Fanuc TP program (LS listing): DISTI_CADC_V5.LS

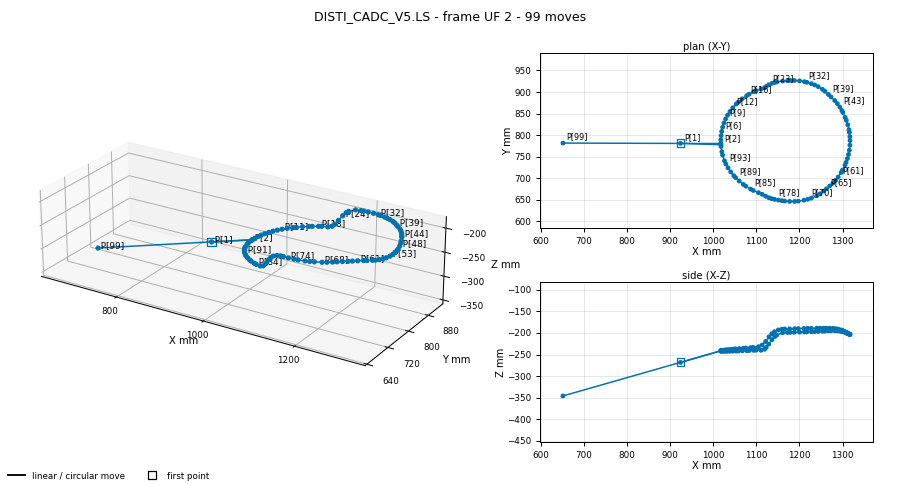
[picture p0: tool path of DISTI_CADC_V5.LS in frame UF 2, 99 of 99 moves have a stored position in this frame; points joined in program order, loops and branches not executed]
/PROG  DISTI_CADC_V5
/ATTR
OWNER		= MNEDITOR;
COMMENT		= "WeldPRO Auto-Gen";
PROG_SIZE	= 7125;
CREATE		= DATE 26-07-30  TIME 16:50:06;
MODIFIED	= DATE 26-07-30  TIME 17:29:32;
FILE_NAME	= DISTI_CA;
VERSION		= 0;
LINE_COUNT	= 113;
MEMORY_SIZE	= 7445;
PROTECT		= READ_WRITE;
TCD:  STACK_SIZE	= 0,
      TASK_PRIORITY	= 50,
      TIME_SLICE	= 0,
      BUSY_LAMP_OFF	= 0,
      ABORT_REQUEST	= 0,
      PAUSE_REQUEST	= 0;
DEFAULT_GROUP	= 1,*,*,*,*;
CONTROL_CODE	= 00000000 00000000;
/APPL
/MN
   1:  !WeldPRO Auto-Generated TPP ;
   2:  !TOR_XL_2026, TOR_xl_2907 ;
   3:   ;
   4:  UFRAME_NUM=2 ;
   5:  UTOOL_NUM=2 ;
   6:  !Feature Approach ;
   7:J P[1] 100% FINE    ;
   8:   ;
   9:  !Segment1 ;
  10:L P[2] 2000mm/sec FINE    ;
  11:   ;
  12:  CALL LASER_OFF    ;
  13:L P[3] R[23:moving]mm/sec CNT100    ;
  14:L P[4] R[23:moving]mm/sec CNT100    ;
  15:L P[5] R[23:moving]mm/sec CNT100    ;
  16:L P[6] R[23:moving]mm/sec CNT100    ;
  17:L P[7] R[23:moving]mm/sec CNT100    ;
  18:L P[8] R[23:moving]mm/sec CNT100    ;
  19:L P[9] R[23:moving]mm/sec CNT100    ;
  20:L P[10] R[23:moving]mm/sec CNT100    ;
  21:L P[11] R[23:moving]mm/sec CNT100    ;
  22:L P[12] R[23:moving]mm/sec CNT100    ;
  23:L P[13] R[23:moving]mm/sec CNT100    ;
  24:L P[14] R[23:moving]mm/sec CNT100    ;
  25:L P[15] R[23:moving]mm/sec CNT100    ;
  26:L P[16] R[23:moving]mm/sec CNT100    ;
  27:L P[17] R[23:moving]mm/sec CNT100    ;
  28:L P[18] R[23:moving]mm/sec CNT100    ;
  29:L P[19] R[23:moving]mm/sec CNT100    ;
  30:L P[20] R[23:moving]mm/sec CNT100    ;
  31:L P[21] R[23:moving]mm/sec CNT100    ;
  32:L P[22] R[23:moving]mm/sec CNT100    ;
  33:L P[23] R[23:moving]mm/sec CNT100    ;
  34:L P[24] R[23:moving]mm/sec CNT100    ;
  35:L P[25] R[23:moving]mm/sec CNT100    ;
  36:L P[26] R[23:moving]mm/sec CNT100    ;
  37:L P[27] R[23:moving]mm/sec CNT100    ;
  38:L P[28] R[23:moving]mm/sec CNT100    ;
  39:L P[29] R[23:moving]mm/sec CNT100    ;
  40:L P[30] R[23:moving]mm/sec CNT100    ;
  41:L P[31] R[23:moving]mm/sec CNT100    ;
  42:L P[32] R[23:moving]mm/sec CNT100    ;
  43:L P[33] R[23:moving]mm/sec CNT100    ;
  44:L P[34] R[23:moving]mm/sec CNT100    ;
  45:L P[35] R[23:moving]mm/sec CNT100    ;
  46:L P[36] R[23:moving]mm/sec CNT100    ;
  47:L P[37] R[23:moving]mm/sec CNT100    ;
  48:L P[38] R[23:moving]mm/sec CNT100    ;
  49:L P[39] R[23:moving]mm/sec CNT100    ;
  50:L P[40] R[23:moving]mm/sec CNT100    ;
  51:L P[41] R[23:moving]mm/sec CNT100    ;
  52:L P[42] R[23:moving]mm/sec CNT100    ;
  53:L P[43] R[23:moving]mm/sec CNT100    ;
  54:L P[44] R[23:moving]mm/sec CNT100    ;
  55:L P[45] R[23:moving]mm/sec CNT100    ;
  56:L P[46] R[23:moving]mm/sec CNT100    ;
  57:L P[47] R[23:moving]mm/sec CNT100    ;
  58:L P[48] R[23:moving]mm/sec CNT100    ;
  59:L P[49] R[23:moving]mm/sec CNT100    ;
  60:L P[50] R[23:moving]mm/sec CNT100    ;
  61:L P[51] R[23:moving]mm/sec CNT100    ;
  62:L P[52] R[23:moving]mm/sec CNT100    ;
  63:L P[53] R[23:moving]mm/sec CNT100    ;
  64:L P[54] R[23:moving]mm/sec CNT100    ;
  65:L P[55] R[23:moving]mm/sec CNT100    ;
  66:L P[56] R[23:moving]mm/sec CNT100    ;
  67:L P[57] R[23:moving]mm/sec CNT100    ;
  68:L P[58] R[23:moving]mm/sec CNT100    ;
  69:L P[59] R[23:moving]mm/sec CNT100    ;
  70:L P[60] R[23:moving]mm/sec CNT100    ;
  71:L P[61] R[23:moving]mm/sec CNT100    ;
  72:L P[62] R[23:moving]mm/sec CNT100    ;
  73:L P[63] R[23:moving]mm/sec CNT100    ;
  74:L P[64] R[23:moving]mm/sec CNT100    ;
  75:L P[65] R[23:moving]mm/sec CNT100    ;
  76:L P[66] R[23:moving]mm/sec CNT100    ;
  77:L P[67] R[23:moving]mm/sec CNT100    ;
  78:L P[68] R[23:moving]mm/sec CNT100    ;
  79:L P[69] R[23:moving]mm/sec CNT100    ;
  80:L P[70] R[23:moving]mm/sec CNT100    ;
  81:L P[71] R[23:moving]mm/sec CNT100    ;
  82:L P[72] R[23:moving]mm/sec CNT100    ;
  83:L P[73] R[23:moving]mm/sec CNT100    ;
  84:L P[74] R[23:moving]mm/sec CNT100    ;
  85:L P[75] R[23:moving]mm/sec CNT100    ;
  86:L P[76] R[23:moving]mm/sec CNT100    ;
  87:L P[77] R[23:moving]mm/sec CNT100    ;
  88:L P[78] R[23:moving]mm/sec CNT100    ;
  89:L P[79] R[23:moving]mm/sec CNT100    ;
  90:L P[80] R[23:moving]mm/sec CNT100    ;
  91:L P[81] R[23:moving]mm/sec CNT100    ;
  92:L P[82] R[23:moving]mm/sec CNT100    ;
  93:L P[83] R[23:moving]mm/sec CNT100    ;
  94:L P[84] R[23:moving]mm/sec CNT100    ;
  95:L P[85] R[23:moving]mm/sec CNT100    ;
  96:L P[86] R[23:moving]mm/sec CNT100    ;
  97:L P[87] R[23:moving]mm/sec CNT100    ;
  98:L P[88] R[23:moving]mm/sec CNT100    ;
  99:L P[89] R[23:moving]mm/sec CNT100    ;
 100:L P[90] R[23:moving]mm/sec CNT100    ;
 101:L P[91] R[23:moving]mm/sec CNT100    ;
 102:L P[92] R[23:moving]mm/sec CNT100    ;
 103:L P[93] R[23:moving]mm/sec CNT100    ;
 104:L P[94] R[23:moving]mm/sec CNT100    ;
 105:L P[95] R[23:moving]mm/sec CNT100    ;
 106:L P[96] R[23:moving]mm/sec CNT100    ;
 107:L P[97] R[23:moving]mm/sec CNT100    ;
 108:L P[98] R[23:moving]mm/sec FINE    ;
 109:  CALL LASER_OFF    ;
 110:   ;
 111:  !Feature Retreat ;
 112:L P[99] 2000mm/sec FINE    ;
 113:  CALL ROTATE    ;
/POS
P[1]{
   GP1:
	UF : 2, UT : 2,		CONFIG : 'F D T, 0, 0, 0',
	X =   924.335  mm,	Y =   780.986  mm,	Z =  -268.284  mm,
	W =  -106.495 deg,	P =   -15.000 deg,	R =    94.234 deg
};
P[2]{
   GP1:
	UF : 2, UT : 2,		CONFIG : 'F D T, 0, 0, 0',
	X =  1018.100  mm,	Y =   777.871  mm,	Z =  -241.295  mm,
	W =  -106.497 deg,	P =   -14.995 deg,	R =    94.216 deg
};
P[3]{
   GP1:
	UF : 2, UT : 2,		CONFIG : 'F D T, 0, 0, 0',
	X =  1017.949  mm,	Y =   780.606  mm,	Z =  -241.391  mm,
	W =  -106.499 deg,	P =   -14.997 deg,	R =    94.226 deg
};
P[4]{
   GP1:
	UF : 2, UT : 2,		CONFIG : 'F D T, 0, 0, 0',
	X =  1017.881  mm,	Y =   789.004  mm,	Z =  -241.645  mm,
	W =  -106.492 deg,	P =   -15.098 deg,	R =    90.372 deg
};
P[5]{
   GP1:
	UF : 2, UT : 2,		CONFIG : 'F D T, 0, 0, 0',
	X =  1018.505  mm,	Y =   798.964  mm,	Z =  -241.908  mm,
	W =  -106.481 deg,	P =   -15.218 deg,	R =    85.605 deg
};
P[6]{
   GP1:
	UF : 2, UT : 2,		CONFIG : 'F D T, 0, 0, 0',
	X =  1019.837  mm,	Y =   808.597  mm,	Z =  -242.115  mm,
	W =  -106.456 deg,	P =   -15.335 deg,	R =    80.815 deg
};
P[7]{
   GP1:
	UF : 2, UT : 2,		CONFIG : 'F D T, 0, 0, 0',
	X =  1022.039  mm,	Y =   818.579  mm,	Z =  -242.280  mm,
	W =  -106.423 deg,	P =   -15.450 deg,	R =    76.090 deg
};
P[8]{
   GP1:
	UF : 2, UT : 2,		CONFIG : 'F D T, 0, 0, 0',
	X =  1025.052  mm,	Y =   828.219  mm,	Z =  -242.385  mm,
	W =  -106.378 deg,	P =   -15.565 deg,	R =    71.217 deg
};
P[9]{
   GP1:
	UF : 2, UT : 2,		CONFIG : 'F D T, 0, 0, 0',
	X =  1028.881  mm,	Y =   837.505  mm,	Z =  -242.427  mm,
	W =  -106.322 deg,	P =   -15.679 deg,	R =    66.207 deg
};
P[10]{
   GP1:
	UF : 2, UT : 2,		CONFIG : 'F D T, 0, 0, 0',
	X =  1033.533  mm,	Y =   846.438  mm,	Z =  -242.409  mm,
	W =  -106.254 deg,	P =   -15.791 deg,	R =    61.015 deg
};
P[11]{
   GP1:
	UF : 2, UT : 2,		CONFIG : 'F D T, 0, 0, 0',
	X =  1038.975  mm,	Y =   854.961  mm,	Z =  -242.328  mm,
	W =  -106.177 deg,	P =   -15.894 deg,	R =    55.979 deg
};
P[12]{
   GP1:
	UF : 2, UT : 2,		CONFIG : 'F D T, 0, 0, 0',
	X =  1045.527  mm,	Y =   863.473  mm,	Z =  -242.178  mm,
	W =  -106.096 deg,	P =   -15.986 deg,	R =    51.162 deg
};
P[13]{
   GP1:
	UF : 2, UT : 2,		CONFIG : 'F D T, 0, 0, 0',
	X =  1053.550  mm,	Y =   872.150  mm,	Z =  -241.942  mm,
	W =  -106.012 deg,	P =   -16.066 deg,	R =    46.632 deg
};
P[14]{
   GP1:
	UF : 2, UT : 2,		CONFIG : 'F D T, 0, 0, 0',
	X =  1058.278  mm,	Y =   876.579  mm,	Z =  -241.784  mm,
	W =  -105.919 deg,	P =   -16.142 deg,	R =    41.952 deg
};
P[15]{
   GP1:
	UF : 2, UT : 2,		CONFIG : 'F D T, 0, 0, 0',
	X =  1067.621  mm,	Y =   884.365  mm,	Z =  -241.434  mm,
	W =  -105.870 deg,	P =   -16.177 deg,	R =    39.609 deg
};
P[16]{
   GP1:
	UF : 2, UT : 2,		CONFIG : 'F D T, 0, 0, 0',
	X =  1077.833  mm,	Y =   891.592  mm,	Z =  -241.014  mm,
	W =  -105.777 deg,	P =   -16.235 deg,	R =    35.365 deg
};
P[17]{
   GP1:
	UF : 2, UT : 2,		CONFIG : 'F D T, 0, 0, 0',
	X =  1083.331  mm,	Y =   894.952  mm,	Z =  -240.778  mm,
	W =  -105.677 deg,	P =   -16.289 deg,	R =    30.964 deg
};
P[18]{
   GP1:
	UF : 2, UT : 2,		CONFIG : 'F D T, 0, 0, 0',
	X =  1094.066  mm,	Y =   900.628  mm,	Z =  -240.278  mm,
	W =  -105.579 deg,	P =   -16.333 deg,	R =    26.830 deg
};
P[19]{
   GP1:
	UF : 2, UT : 2,		CONFIG : 'F D T, 0, 0, 0',
	X =  1099.603  mm,	Y =   903.126  mm,	Z =  -240.005  mm,
	W =  -105.536 deg,	P =   -16.344 deg,	R =    25.018 deg
};
P[20]{
   GP1:
	UF : 2, UT : 2,		CONFIG : 'F D T, 0, 0, 0',
	X =  1111.079  mm,	Y =   907.027  mm,	Z =  -240.106  mm,
	W =  -116.027 deg,	P =   -16.063 deg,	R =    30.267 deg
};
P[21]{
   GP1:
	UF : 2, UT : 2,		CONFIG : 'F D T, 0, 0, 0',
	X =  1119.171  mm,	Y =   909.914  mm,	Z =  -237.723  mm,
	W =  -126.877 deg,	P =   -15.356 deg,	R =    25.893 deg
};
P[22]{
   GP1:
	UF : 2, UT : 2,		CONFIG : 'F D T, 0, 0, 0',
	X =  1122.964  mm,	Y =   912.740  mm,	Z =  -233.580  mm,
	W =  -119.393 deg,	P =   -15.981 deg,	R =    16.221 deg
};
P[23]{
   GP1:
	UF : 2, UT : 2,		CONFIG : 'F D T, 0, 0, 0',
	X =  1128.743  mm,	Y =   916.697  mm,	Z =  -225.925  mm,
	W =  -115.329 deg,	P =   -16.208 deg,	R =    11.788 deg
};
P[24]{
   GP1:
	UF : 2, UT : 2,		CONFIG : 'F D T, 0, 0, 0',
	X =  1136.345  mm,	Y =   920.133  mm,	Z =  -215.586  mm,
	W =  -112.639 deg,	P =   -16.315 deg,	R =     9.714 deg
};
P[25]{
   GP1:
	UF : 2, UT : 2,		CONFIG : 'F D T, 0, 0, 0',
	X =  1142.709  mm,	Y =   922.174  mm,	Z =  -208.396  mm,
	W =  -110.015 deg,	P =   -16.386 deg,	R =     9.649 deg
};
P[26]{
   GP1:
	UF : 2, UT : 2,		CONFIG : 'F D T, 0, 0, 0',
	X =  1147.389  mm,	Y =   923.274  mm,	Z =  -204.928  mm,
	W =  -108.552 deg,	P =   -16.418 deg,	R =     8.950 deg
};
P[27]{
   GP1:
	UF : 2, UT : 2,		CONFIG : 'F D T, 0, 0, 0',
	X =  1161.068  mm,	Y =   925.459  mm,	Z =  -199.565  mm,
	W =  -105.409 deg,	P =   -16.443 deg,	R =     6.805 deg
};
P[28]{
   GP1:
	UF : 2, UT : 2,		CONFIG : 'F D T, 0, 0, 0',
	X =  1172.554  mm,	Y =   926.477  mm,	Z =  -198.839  mm,
	W =  -104.866 deg,	P =   -16.444 deg,	R =     5.597 deg
};
P[29]{
   GP1:
	UF : 2, UT : 2,		CONFIG : 'F D T, 0, 0, 0',
	X =  1178.771  mm,	Y =   926.778  mm,	Z =  -198.674  mm,
	W =  -104.887 deg,	P =   -16.444 deg,	R =     3.523 deg
};
P[30]{
   GP1:
	UF : 2, UT : 2,		CONFIG : 'F D T, 0, 0, 0',
	X =  1188.194  mm,	Y =   926.816  mm,	Z =  -198.418  mm,
	W =  -104.930 deg,	P =   -16.439 deg,	R =     -.728 deg
};
P[31]{
   GP1:
	UF : 2, UT : 2,		CONFIG : 'F D T, 0, 0, 0',
	X =  1200.286  mm,	Y =   925.904  mm,	Z =  -198.059  mm,
	W =  -104.979 deg,	P =   -16.424 deg,	R =    -5.541 deg
};
P[32]{
   GP1:
	UF : 2, UT : 2,		CONFIG : 'F D T, 0, 0, 0',
	X =  1211.474  mm,	Y =   923.979  mm,	Z =  -197.695  mm,
	W =  -105.028 deg,	P =   -16.400 deg,	R =   -10.259 deg
};
P[33]{
   GP1:
	UF : 2, UT : 2,		CONFIG : 'F D T, 0, 0, 0',
	X =  1217.339  mm,	Y =   922.538  mm,	Z =  -197.505  mm,
	W =  -105.070 deg,	P =   -16.371 deg,	R =   -14.490 deg
};
P[34]{
   GP1:
	UF : 2, UT : 2,		CONFIG : 'F D T, 0, 0, 0',
	X =  1227.782  mm,	Y =   919.324  mm,	Z =  -197.120  mm,
	W =  -105.112 deg,	P =   -16.334 deg,	R =   -18.515 deg
};
P[35]{
   GP1:
	UF : 2, UT : 2,		CONFIG : 'F D T, 0, 0, 0',
	X =  1235.361  mm,	Y =   916.374  mm,	Z =  -196.835  mm,
	W =  -105.158 deg,	P =   -16.285 deg,	R =   -23.051 deg
};
P[36]{
   GP1:
	UF : 2, UT : 2,		CONFIG : 'F D T, 0, 0, 0',
	X =  1243.527  mm,	Y =   912.450  mm,	Z =  -196.518  mm,
	W =  -105.219 deg,	P =   -16.204 deg,	R =   -29.417 deg
};
P[37]{
   GP1:
	UF : 2, UT : 2,		CONFIG : 'F D T, 0, 0, 0',
	X =  1253.417  mm,	Y =   906.235  mm,	Z =  -196.108  mm,
	W =  -105.311 deg,	P =   -16.047 deg,	R =   -39.415 deg
};
P[38]{
   GP1:
	UF : 2, UT : 2,		CONFIG : 'F D T, 0, 0, 0',
	X =  1259.200  mm,	Y =   901.667  mm,	Z =  -195.783  mm,
	W =  -105.307 deg,	P =   -16.055 deg,	R =   -38.974 deg
};
P[39]{
   GP1:
	UF : 2, UT : 2,		CONFIG : 'F D T, 0, 0, 0',
	X =  1267.291  mm,	Y =   894.227  mm,	Z =  -195.295  mm,
	W =  -105.302 deg,	P =   -16.063 deg,	R =   -38.625 deg
};
P[40]{
   GP1:
	UF : 2, UT : 2,		CONFIG : 'F D T, 0, 0, 0',
	X =  1273.355  mm,	Y =   888.496  mm,	Z =  -195.066  mm,
	W =  -105.469 deg,	P =   -15.944 deg,	R =   -44.976 deg
};
P[41]{
   GP1:
	UF : 2, UT : 2,		CONFIG : 'F D T, 0, 0, 0',
	X =  1281.920  mm,	Y =   880.180  mm,	Z =  -194.951  mm,
	W =  -105.661 deg,	P =   -15.890 deg,	R =   -47.714 deg
};
P[42]{
   GP1:
	UF : 2, UT : 2,		CONFIG : 'F D T, 0, 0, 0',
	X =  1287.931  mm,	Y =   873.124  mm,	Z =  -195.180  mm,
	W =  -106.210 deg,	P =   -15.792 deg,	R =   -52.259 deg
};
P[43]{
   GP1:
	UF : 2, UT : 2,		CONFIG : 'F D T, 0, 0, 0',
	X =  1293.538  mm,	Y =   865.209  mm,	Z =  -195.720  mm,
	W =  -106.927 deg,	P =   -15.688 deg,	R =   -56.663 deg
};
P[44]{
   GP1:
	UF : 2, UT : 2,		CONFIG : 'F D T, 0, 0, 0',
	X =  1298.359  mm,	Y =   857.230  mm,	Z =  -196.540  mm,
	W =  -107.603 deg,	P =   -15.597 deg,	R =   -60.243 deg
};
P[45]{
   GP1:
	UF : 2, UT : 2,		CONFIG : 'F D T, 0, 0, 0',
	X =  1300.727  mm,	Y =   852.739  mm,	Z =  -197.136  mm,
	W =  -108.271 deg,	P =   -15.504 deg,	R =   -63.685 deg
};
P[46]{
   GP1:
	UF : 2, UT : 2,		CONFIG : 'F D T, 0, 0, 0',
	X =  1306.110  mm,	Y =   841.187  mm,	Z =  -199.012  mm,
	W =  -109.144 deg,	P =   -15.377 deg,	R =   -68.203 deg
};
P[47]{
   GP1:
	UF : 2, UT : 2,		CONFIG : 'F D T, 0, 0, 0',
	X =  1308.723  mm,	Y =   834.365  mm,	Z =  -200.199  mm,
	W =  -109.899 deg,	P =   -15.253 deg,	R =   -72.505 deg
};
P[48]{
   GP1:
	UF : 2, UT : 2,		CONFIG : 'F D T, 0, 0, 0',
	X =  1312.088  mm,	Y =   824.073  mm,	Z =  -201.668  mm,
	W =  -110.273 deg,	P =   -15.181 deg,	R =   -74.981 deg
};
P[49]{
   GP1:
	UF : 2, UT : 2,		CONFIG : 'F D T, 0, 0, 0',
	X =  1314.829  mm,	Y =   812.726  mm,	Z =  -202.833  mm,
	W =  -110.635 deg,	P =   -14.305 deg,	R =   -78.232 deg
};
P[50]{
   GP1:
	UF : 2, UT : 2,		CONFIG : 'F D T, 0, 0, 0',
	X =  1315.830  mm,	Y =   806.528  mm,	Z =  -203.260  mm,
	W =  -111.054 deg,	P =   -14.769 deg,	R =   -83.164 deg
};
P[51]{
   GP1:
	UF : 2, UT : 2,		CONFIG : 'F D T, 0, 0, 0',
	X =  1316.913  mm,	Y =   796.538  mm,	Z =  -203.641  mm,
	W =  -111.190 deg,	P =   -15.305 deg,	R =   -88.308 deg
};
P[52]{
   GP1:
	UF : 2, UT : 2,		CONFIG : 'F D T, 0, 0, 0',
	X =  1317.315  mm,	Y =   787.558  mm,	Z =  -203.666  mm,
	W =  -111.129 deg,	P =   -15.645 deg,	R =   -91.614 deg
};
P[53]{
   GP1:
	UF : 2, UT : 2,		CONFIG : 'F D T, 0, 0, 0',
	X =  1317.000  mm,	Y =   776.840  mm,	Z =  -203.309  mm,
	W =  -110.757 deg,	P =   -14.624 deg,	R =   -96.575 deg
};
P[54]{
   GP1:
	UF : 2, UT : 2,		CONFIG : 'F D T, 0, 0, 0',
	X =  1315.687  mm,	Y =   765.039  mm,	Z =  -202.411  mm,
	W =  -110.276 deg,	P =   -14.535 deg,	R =  -100.836 deg
};
P[55]{
   GP1:
	UF : 2, UT : 2,		CONFIG : 'F D T, 0, 0, 0',
	X =  1313.778  mm,	Y =   755.222  mm,	Z =  -201.256  mm,
	W =  -109.635 deg,	P =   -14.447 deg,	R =  -105.265 deg
};
P[56]{
   GP1:
	UF : 2, UT : 2,		CONFIG : 'F D T, 0, 0, 0',
	X =  1311.241  mm,	Y =   745.826  mm,	Z =  -199.809  mm,
	W =  -109.083 deg,	P =   -14.382 deg,	R =  -108.625 deg
};
P[57]{
   GP1:
	UF : 2, UT : 2,		CONFIG : 'F D T, 0, 0, 0',
	X =  1308.150  mm,	Y =   736.915  mm,	Z =  -198.124  mm,
	W =  -108.349 deg,	P =   -14.302 deg,	R =  -112.873 deg
};
P[58]{
   GP1:
	UF : 2, UT : 2,		CONFIG : 'F D T, 0, 0, 0',
	X =  1305.598  mm,	Y =   730.728  mm,	Z =  -196.774  mm,
	W =  -107.748 deg,	P =   -14.239 deg,	R =  -116.265 deg
};
P[59]{
   GP1:
	UF : 2, UT : 2,		CONFIG : 'F D T, 0, 0, 0',
	X =  1299.951  mm,	Y =   719.236  mm,	Z =  -193.996  mm,
	W =  -106.927 deg,	P =   -14.148 deg,	R =  -121.193 deg
};
P[60]{
   GP1:
	UF : 2, UT : 2,		CONFIG : 'F D T, 0, 0, 0',
	X =  1296.675  mm,	Y =   713.566  mm,	Z =  -192.788  mm,
	W =  -106.269 deg,	P =   -14.066 deg,	R =  -125.698 deg
};
P[61]{
   GP1:
	UF : 2, UT : 2,		CONFIG : 'F D T, 0, 0, 0',
	X =  1289.858  mm,	Y =   703.173  mm,	Z =  -190.968  mm,
	W =  -105.781 deg,	P =   -13.988 deg,	R =  -130.143 deg
};
P[62]{
   GP1:
	UF : 2, UT : 2,		CONFIG : 'F D T, 0, 0, 0',
	X =  1283.513  mm,	Y =   695.116  mm,	Z =  -189.944  mm,
	W =  -105.527 deg,	P =   -13.913 deg,	R =  -134.519 deg
};
P[63]{
   GP1:
	UF : 2, UT : 2,		CONFIG : 'F D T, 0, 0, 0',
	X =  1277.726  mm,	Y =   688.980  mm,	Z =  -189.402  mm,
	W =  -105.437 deg,	P =   -13.849 deg,	R =  -138.629 deg
};
P[64]{
   GP1:
	UF : 2, UT : 2,		CONFIG : 'F D T, 0, 0, 0',
	X =  1270.076  mm,	Y =   682.016  mm,	Z =  -189.027  mm,
	W =  -105.429 deg,	P =   -13.831 deg,	R =  -139.837 deg
};
P[65]{
   GP1:
	UF : 2, UT : 2,		CONFIG : 'F D T, 0, 0, 0',
	X =  1262.526  mm,	Y =   675.566  mm,	Z =  -188.929  mm,
	W =  -105.443 deg,	P =   -13.863 deg,	R =  -137.727 deg
};
P[66]{
   GP1:
	UF : 2, UT : 2,		CONFIG : 'F D T, 0, 0, 0',
	X =  1256.210  mm,	Y =   670.346  mm,	Z =  -188.936  mm,
	W =  -105.373 deg,	P =   -13.729 deg,	R =  -147.436 deg
};
P[67]{
   GP1:
	UF : 2, UT : 2,		CONFIG : 'F D T, 0, 0, 0',
	X =  1247.902  mm,	Y =   664.235  mm,	Z =  -188.960  mm,
	W =  -105.298 deg,	P =   -13.637 deg,	R =  -156.529 deg
};
P[68]{
   GP1:
	UF : 2, UT : 2,		CONFIG : 'F D T, 0, 0, 0',
	X =  1240.286  mm,	Y =   659.590  mm,	Z =  -189.026  mm,
	W =  -105.277 deg,	P =   -13.618 deg,	R =  -158.976 deg
};
P[69]{
   GP1:
	UF : 2, UT : 2,		CONFIG : 'F D T, 0, 0, 0',
	X =  1227.578  mm,	Y =   654.053  mm,	Z =  -189.213  mm,
	W =  -105.241 deg,	P =   -13.592 deg,	R =  -162.969 deg
};
P[70]{
   GP1:
	UF : 2, UT : 2,		CONFIG : 'F D T, 0, 0, 0',
	X =  1219.295  mm,	Y =   651.430  mm,	Z =  -189.358  mm,
	W =  -105.203 deg,	P =   -13.573 deg,	R =  -167.022 deg
};
P[71]{
   GP1:
	UF : 2, UT : 2,		CONFIG : 'F D T, 0, 0, 0',
	X =  1210.620  mm,	Y =   649.289  mm,	Z =  -189.525  mm,
	W =  -105.159 deg,	P =   -13.560 deg,	R =  -171.569 deg
};
P[72]{
   GP1:
	UF : 2, UT : 2,		CONFIG : 'F D T, 0, 0, 0',
	X =  1197.379  mm,	Y =   647.095  mm,	Z =  -189.828  mm,
	W =  -105.113 deg,	P =   -13.556 deg,	R =  -176.312 deg
};
P[73]{
   GP1:
	UF : 2, UT : 2,		CONFIG : 'F D T, 0, 0, 0',
	X =  1188.999  mm,	Y =   646.477  mm,	Z =  -190.033  mm,
	W =  -105.068 deg,	P =   -13.561 deg,	R =   179.213 deg
};
P[74]{
   GP1:
	UF : 2, UT : 2,		CONFIG : 'F D T, 0, 0, 0',
	X =  1177.274  mm,	Y =   646.506  mm,	Z =  -190.367  mm,
	W =  -105.038 deg,	P =   -13.569 deg,	R =   176.231 deg
};
P[75]{
   GP1:
	UF : 2, UT : 2,		CONFIG : 'F D T, 0, 0, 0',
	X =  1165.873  mm,	Y =   647.395  mm,	Z =  -190.762  mm,
	W =  -105.207 deg,	P =   -13.572 deg,	R =   175.290 deg
};
P[76]{
   GP1:
	UF : 2, UT : 2,		CONFIG : 'F D T, 0, 0, 0',
	X =  1159.530  mm,	Y =   648.231  mm,	Z =  -191.266  mm,
	W =  -107.012 deg,	P =   -13.569 deg,	R =   174.537 deg
};
P[77]{
   GP1:
	UF : 2, UT : 2,		CONFIG : 'F D T, 0, 0, 0',
	X =  1151.090  mm,	Y =   649.552  mm,	Z =  -192.887  mm,
	W =  -109.414 deg,	P =   -13.538 deg,	R =   174.483 deg
};
P[78]{
   GP1:
	UF : 2, UT : 2,		CONFIG : 'F D T, 0, 0, 0',
	X =  1142.165  mm,	Y =   651.267  mm,	Z =  -196.994  mm,
	W =  -112.196 deg,	P =   -13.466 deg,	R =   175.323 deg
};
P[79]{
   GP1:
	UF : 2, UT : 2,		CONFIG : 'F D T, 0, 0, 0',
	X =  1135.832  mm,	Y =   652.821  mm,	Z =  -201.869  mm,
	W =  -114.872 deg,	P =   -13.369 deg,	R =   175.422 deg
};
P[80]{
   GP1:
	UF : 2, UT : 2,		CONFIG : 'F D T, 0, 0, 0',
	X =  1129.472  mm,	Y =   654.941  mm,	Z =  -208.996  mm,
	W =  -120.114 deg,	P =   -13.109 deg,	R =   172.293 deg
};
P[81]{
   GP1:
	UF : 2, UT : 2,		CONFIG : 'F D T, 0, 0, 0',
	X =  1121.646  mm,	Y =   658.652  mm,	Z =  -219.868  mm,
	W =  -126.810 deg,	P =   -12.622 deg,	R =   167.787 deg
};
P[82]{
   GP1:
	UF : 2, UT : 2,		CONFIG : 'F D T, 0, 0, 0',
	X =  1113.631  mm,	Y =   662.962  mm,	Z =  -227.981  mm,
	W =  -119.561 deg,	P =   -13.285 deg,	R =   157.806 deg
};
P[83]{
   GP1:
	UF : 2, UT : 2,		CONFIG : 'F D T, 0, 0, 0',
	X =  1105.134  mm,	Y =   666.653  mm,	Z =  -231.760  mm,
	W =  -107.219 deg,	P =   -13.741 deg,	R =   154.408 deg
};
P[84]{
   GP1:
	UF : 2, UT : 2,		CONFIG : 'F D T, 0, 0, 0',
	X =  1093.094  mm,	Y =   671.827  mm,	Z =  -233.397  mm,
	W =  -105.746 deg,	P =   -13.749 deg,	R =   154.142 deg
};
P[85]{
   GP1:
	UF : 2, UT : 2,		CONFIG : 'F D T, 0, 0, 0',
	X =  1086.938  mm,	Y =   674.999  mm,	Z =  -233.893  mm,
	W =  -105.804 deg,	P =   -13.784 deg,	R =   151.506 deg
};
P[86]{
   GP1:
	UF : 2, UT : 2,		CONFIG : 'F D T, 0, 0, 0',
	X =  1075.720  mm,	Y =   681.824  mm,	Z =  -234.827  mm,
	W =  -105.885 deg,	P =   -13.838 deg,	R =   147.739 deg
};
P[87]{
   GP1:
	UF : 2, UT : 2,		CONFIG : 'F D T, 0, 0, 0',
	X =  1070.116  mm,	Y =   685.851  mm,	Z =  -235.283  mm,
	W =  -105.988 deg,	P =   -13.918 deg,	R =   142.681 deg
};
P[88]{
   GP1:
	UF : 2, UT : 2,		CONFIG : 'F D T, 0, 0, 0',
	X =  1060.382  mm,	Y =   693.768  mm,	Z =  -236.124  mm,
	W =  -106.082 deg,	P =   -14.006 deg,	R =   137.688 deg
};
P[89]{
   GP1:
	UF : 2, UT : 2,		CONFIG : 'F D T, 0, 0, 0',
	X =  1051.934  mm,	Y =   701.724  mm,	Z =  -236.861  mm,
	W =  -106.129 deg,	P =   -14.056 deg,	R =   135.015 deg
};
P[90]{
   GP1:
	UF : 2, UT : 2,		CONFIG : 'F D T, 0, 0, 0',
	X =  1047.883  mm,	Y =   706.090  mm,	Z =  -237.237  mm,
	W =  -106.186 deg,	P =   -14.117 deg,	R =   131.622 deg
};
P[91]{
   GP1:
	UF : 2, UT : 2,		CONFIG : 'F D T, 0, 0, 0',
	X =  1040.744  mm,	Y =   714.877  mm,	Z =  -237.970  mm,
	W =  -106.269 deg,	P =   -14.239 deg,	R =   125.999 deg
};
P[92]{
   GP1:
	UF : 2, UT : 2,		CONFIG : 'F D T, 0, 0, 0',
	X =  1034.468  mm,	Y =   724.256  mm,	Z =  -238.645  mm,
	W =  -106.343 deg,	P =   -14.367 deg,	R =   120.225 deg
};
P[93]{
   GP1:
	UF : 2, UT : 2,		CONFIG : 'F D T, 0, 0, 0',
	X =  1029.612  mm,	Y =   733.175  mm,	Z =  -239.197  mm,
	W =  -106.384 deg,	P =   -14.458 deg,	R =   116.261 deg
};
P[94]{
   GP1:
	UF : 2, UT : 2,		CONFIG : 'F D T, 0, 0, 0',
	X =  1026.316  mm,	Y =   740.635  mm,	Z =  -239.610  mm,
	W =  -106.433 deg,	P =   -14.556 deg,	R =   111.957 deg
};
P[95]{
   GP1:
	UF : 2, UT : 2,		CONFIG : 'F D T, 0, 0, 0',
	X =  1021.946  mm,	Y =   753.812  mm,	Z =  -240.308  mm,
	W =  -106.465 deg,	P =   -14.714 deg,	R =   105.666 deg
};
P[96]{
   GP1:
	UF : 2, UT : 2,		CONFIG : 'F D T, 0, 1, 0',
	X =  1020.133  mm,	Y =   761.720  mm,	Z =  -240.690  mm,
	W =  -106.480 deg,	P =   -14.798 deg,	R =   102.261 deg
};
P[97]{
   GP1:
	UF : 2, UT : 2,		CONFIG : 'F D T, 0, 1, 0',
	X =  1018.418  mm,	Y =   773.701  mm,	Z =  -241.160  mm,
	W =  -106.494 deg,	P =   -14.935 deg,	R =    96.827 deg
};
P[98]{
   GP1:
	UF : 2, UT : 2,		CONFIG : 'F D T, 0, 1, 0',
	X =  1017.949  mm,	Y =   780.604  mm,	Z =  -241.391  mm,
	W =  -106.501 deg,	P =   -15.000 deg,	R =    94.236 deg
};
P[99]{
   GP1:
	UF : 2, UT : 2,		CONFIG : 'F D T, 0, 1, 0',
	X =   651.995  mm,	Y =   781.694  mm,	Z =  -345.952  mm,
	W =  -106.495 deg,	P =   -15.000 deg,	R =    94.234 deg
};
/END
